INTERFACE I_ServerResponse

METHOD PUBLIC Accepted
VAR_INPUT
END_VAR
END_METHOD

METHOD PUBLIC Busy
VAR_INPUT
END_VAR
END_METHOD

METHOD PUBLIC Error
VAR_INPUT
	Message : T_MAXSTRING;
END_VAR
END_METHOD

PROPERTY PUBLIC Header : I_Header
GET
END_GET
END_PROPERTY

PROPERTY PUBLIC HeadersSent : BOOL
GET
END_GET
END_PROPERTY

METHOD PUBLIC Pending
VAR_INPUT
	ResponseId : REFERENCE TO T_MAXSTRING;
	RetryDelayInMs : UDINT;
END_VAR
END_METHOD

METHOD PUBLIC Success
VAR_INPUT
END_VAR
END_METHOD

METHOD PUBLIC SuccessWithPayload
VAR_INPUT
	PayloadDataAddress : PVOID;
	PayloadDataSize : UDINT;
END_VAR
END_METHOD

END_INTERFACE

(* stored: Version 1.1.0.1, ProductVersion 3.1.4024.12
   Itf I_ServerResponse: Id {e40a3331-8557-094a-10a6-a8155fda0cd7}
   Method Accepted: Id {f50cccf4-f9bd-06f6-2a09-f50e48c83f8e}
   Method Busy: Id {2510a061-c35e-00b3-03db-2bc618421e85}
   Method Error: Id {457d175b-7c57-09cf-2d6a-81bb7a2d9875}
   Property Header: Id {18b6640e-6fe8-0c08-3f00-501baa1837ec}
   Get Get: Id {69dcb55f-a337-0aeb-00b0-5925e28f5a31}
   Property HeadersSent: Id {fe5f2030-992b-0c19-33b4-53749d4c7c11}
   Get Get: Id {e0842237-f2ab-0ae7-14af-4777f0154a29}
   Method Pending: Id {95467046-a172-01c8-3341-28dc1b8903c9}
   Method Success: Id {5ae10595-e0eb-0002-1860-1a946943d841}
   Method SuccessWithPayload: Id {470d5faa-cb78-00b4-1128-929187ae46da} *)
